FUNCTION_BLOCK Request_F (* Template for a Basic Function Block Type *)
  (* Standard: 61499-2 *)
  (* Version 1.0, 2022-01-17, Fan *)
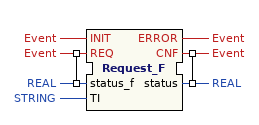
  EVENT_INPUT
    INIT; (* Initialization Request *)
    REQ WITH status_f; (* Normal Execution Request *)
  END_EVENT
  EVENT_OUTPUT
    ERROR; (* Initialization Confirm *)
    CNF WITH status; (* Execution Confirmation *)
  END_EVENT
  VAR_INPUT
    status_f : REAL; (* Input event qualifier *)
    TI : STRING;
  END_VAR
  VAR_OUTPUT
    status : REAL; (* Output event qualifier *)
  END_VAR
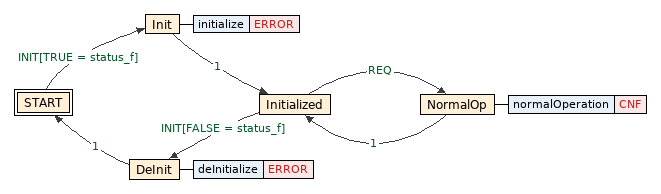
  EC_STATES
    START; (* Initial State *)
    Init : initialize -> ERROR; (* Initialization *)
    NormalOp : normalOperation -> CNF; (* Normal execution *)
    Initialized;
    DeInit : deInitialize -> ERROR;
  END_STATES
  EC_TRANSITIONS
    START TO Init := INIT[TRUE = status_f];
    Init TO Initialized := 1;
    Initialized TO NormalOp := REQ;
    NormalOp TO Initialized := 1;
    DeInit TO START := 1;
    Initialized TO DeInit := INIT[FALSE = status_f];
  END_TRANSITIONS
  ALGORITHM initialize IN ST: (* Initialization algorithm *)

  END_ALGORITHM
  ALGORITHM deInitialize IN ST: (* Normally executed algorithm *)

  END_ALGORITHM
  ALGORITHM normalOperation IN ST: (* new algorithm *)

  END_ALGORITHM
END_FUNCTION_BLOCK
